# EPICS autosave request: ADApp/Db/NDROI_settings.req
$(P)$(R)Name
$(P)$(R)DataTypeOut
$(P)$(R)BinX
$(P)$(R)BinY
$(P)$(R)BinZ
$(P)$(R)MinX
$(P)$(R)MinY
$(P)$(R)MinZ
$(P)$(R)SizeX
$(P)$(R)SizeY
$(P)$(R)SizeZ
$(P)$(R)ReverseX
$(P)$(R)ReverseY
$(P)$(R)ReverseZ
$(P)$(R)AutoSizeX
$(P)$(R)AutoSizeY
$(P)$(R)AutoSizeZ
$(P)$(R)EnableX
$(P)$(R)EnableY
$(P)$(R)EnableZ
$(P)$(R)EnableScale
$(P)$(R)Scale
$(P)$(R)CollapseDims
file "NDPluginBase_settings.req", P=$(P), R=$(R)
